ABB RobotStudio station: EGM_Demo.rsstn

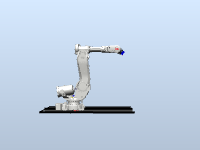
Station EGM_Demo (saved by RobotStudio 6.5.7479.130)
Controller EGM_Demo
  mechanical unit ROB_1: IRB6640_180_255__04, 6 joints, base frame (0, 0, 0) mm
Layout (positions relative to the parent item):
  - IRB6640_180_255__04 [mechanism, from Robots\IRB6640_180_255_G_04.rslib] at (0, 0, 0) mm; joint values [0, 0, 0, 0, 0.5236, 0] (rad or m)
